PROGRAM PB_TestRunner
VAR
    Init : BOOL := TRUE;
END_VAR

IF Init THEN
    TestFramework.TestRunner.AddTestSuite(UnitTests.TestFrameworkTests);
    Init := FALSE;
END_IF

TestFramework.TestRunner(
    RunTestsSequentially := TRUE,
    ManualTestRunsOnly := TRUE);

END_PROGRAM

(* stored: Version 1.1.0.1, ProductVersion 3.1.4024.4
   POU PB_TestRunner: Id {13d7246e-c481-4cd4-9fbf-5e6440dda62d}, SpecialFunc None *)
